(* IEC 61131-3 sources: Stat_Resistant_AI_Coding/src/plc/project/Station010, 9 files *)

(* ---- Wp100ResistanceResultStruct.st ---- *)
{attribute 'OPC.UA.DA.StructuredType':='1'}
TYPE Wp100ResistanceResultStruct :
STRUCT
  /// TRUE after SINGLE_MEAS has completed and the values below have been copied
  Valid      : BOOL;
  OutOfLimit : BOOL;
  Ok         : BOOL;
  Value      : REAL;
  Temperature : REAL;
END_STRUCT
END_TYPE

(* ---- Wp100RunResultStruct.st ---- *)
{attribute 'OPC.UA.DA.StructuredType':='1'}
TYPE Wp100RunResultStruct :
STRUCT
  /// Fixture position requested for this execution
  MeasurePos           : MeasurePsoEnum;
  /// TRUE after the requested position has passed the three-sensor one-hot check
  FixturePositionValid : BOOL;
  /// Burster resistance measurement result
  Resistance           : Wp100ResistanceResultStruct;
  /// Kistler force/stroke measurement result
  Kistler              : Wp100KistlerResultStruct;
END_STRUCT
END_TYPE

(* ---- Wp100RunSequenceResultStruct.st ---- *)
TYPE Wp100RunSequenceResultStruct :
STRUCT
  /// Result captured after the left-position atomic measurement
  Left   : Wp100RunResultStruct;
  /// Result captured after the middle-position atomic measurement
  Middle : Wp100RunResultStruct;
  /// Result captured after the right-position atomic measurement
  Right  : Wp100RunResultStruct;
END_STRUCT
END_TYPE

(* ---- AiForceTrace.gvl.st ---- *)
{attribute 'qualified_only'}
VAR_GLOBAL
  Recorder : FB_HmiForceTrace;
END_VAR

(* ---- AiWp100.gvl.st ---- *)
{attribute 'qualified_only'}
VAR_GLOBAL
  BursterProgramSelect : FB_Wp100BursterProgramSelect;
END_VAR

(* ---- FB_HmiForceTrace.st ---- *)
(* ===== OBJECT FB_HmiForceTrace ===== *)
(* ===== DECLARATION ===== *)
FUNCTION_BLOCK FB_HmiForceTrace
VAR_INPUT
  Measuring : BOOL;
  QualityGood : BOOL;
  ForceN : REAL;
END_VAR
VAR_OUTPUT
  LeftFrame : ARRAY [0..30035] OF DWORD;
  MiddleFrame : ARRAY [0..30035] OF DWORD;
  RightFrame : ARRAY [0..30035] OF DWORD;
  StatisticsFrame : ARRAY [0..209] OF DWORD;
  Published : BOOL;
  PublishedPosition : UDINT;
  Cleared : BOOL;
  Qualified : BOOL;
  DataGood : BOOL;
  SampleTime : UDINT;
END_VAR
VAR
  _stats : FB_PressForceStatistics;
  _trace : ARRAY [1..3] OF T_HmiForceBuffer;
  _stat : ARRAY [1..3,0..63] OF DWORD;
  _payloadHash : ARRAY [1..3] OF UDINT;
  _frozen : ARRAY [1..3] OF BOOL;
  _configured : BOOL;
  _guardActive : BOOL;
  _clearPending : BOOL;
  _urgent : BOOL;
  _initialized : BOOL;
  _normalEndRequested : BOOL;
  _threshold : REAL;
  _limit : REAL;
  _window : UDINT;
  _timeout : UDINT;
  _now : UDINT;
  _started : UDINT;
  _elapsed : UDINT;
  _lastSample : UDINT;
  _lastPublish : UDINT;
  _boot : UDINT;
  _cycle : UDINT;
  _acquisition : UDINT;
  _sequence : UDINT;
  _scan : UDINT;
  _sampledScan : UDINT;
  _position : UDINT;
  _state : UDINT;
  _hash : UDINT;
  _word : U_HmiForceWord;
  _p : DINT;
  _i : DINT;
  _j : DINT;
END_VAR
(* ===== IMPLEMENTATION ===== *)
// MainTask caller. HMI timing never owns acquisition or process decisions.
_now := TIME_TO_UDINT(TIME());
_scan := _scan + 1;
Published := FALSE;
Cleared := _clearPending;
_clearPending := FALSE;
IF ( NOT _initialized )
THEN
  _initialized := TRUE;
  _boot := _now;
  _urgent := TRUE;
END_IF
IF ( _state = 1 )
THEN
  IF ( NOT _guardActive )
  THEN
    Sample(ValueN := ForceN, Healthy := QualityGood, AtWork := FALSE);
  ELSIF ( ( _now - _lastSample ) > 15 )
  THEN
    // Missing cyclic guard calls must not leave a stale TRUE for the next DONE.
    DataGood := FALSE;
    Qualified := FALSE;
  END_IF
  IF ( NOT QualityGood ) OR ( NOT ( ForceN = ForceN ) ) OR
     ( ABS(ForceN) > REAL#3.402823E38 )
  THEN
    Finish(Reason := 5, LastForceN := ForceN);
  ELSIF ( NOT Measuring )
  THEN
    IF ( _normalEndRequested )
    THEN
      Finish(Reason := 2, LastForceN := ForceN);
    ELSE
      Finish(Reason := 5, LastForceN := ForceN);
    END_IF
  END_IF
END_IF
IF ( _urgent ) OR ( ( _now - _lastPublish ) >= 100 ) OR ( Cleared )
THEN
  Publish();
END_IF

(* ===== OBJECT Configure ===== *)
(* ===== DECLARATION ===== *)
METHOD PUBLIC Configure
VAR_INPUT
  ThresholdN : REAL;
  LimitN : REAL;
  WindowMs : UDINT;
  TimeoutMs : UDINT;
END_VAR
(* ===== IMPLEMENTATION ===== *)
// Once per position, before Kistler START. Changes take effect next position.
_threshold := ThresholdN;
_limit := LimitN;
_window := WindowMs;
_timeout := TimeoutMs;
_configured := TRUE;

(* ===== OBJECT BeginCycle ===== *)
(* ===== DECLARATION ===== *)
METHOD PUBLIC BeginCycle
(* ===== IMPLEMENTATION ===== *)
_cycle := _cycle + 1;
IF ( _cycle = 0 )
THEN
  _cycle := 1;
END_IF
// Only Count is authoritative. Old payload beyond Count is never displayed.
FOR _p := 1 TO 3 DO
  FOR _i := 0 TO 31 DO
    _trace[_p][_i] := 0;
  END_FOR
  FOR _i := 0 TO 63 DO
    _stat[_p,_i] := 0;
  END_FOR
  _trace[_p][1] := DWORD#2;
  _trace[_p][3] := UDINT_TO_DWORD(_cycle);
  _trace[_p][5] := DINT_TO_DWORD(_p);
  _trace[_p][16] := DWORD#6;
  _payloadHash[_p] := UDINT#2166136261;
  _frozen[_p] := FALSE;
END_FOR
_position := 0;
_state := 0;
_configured := FALSE;
_guardActive := FALSE;
Qualified := FALSE;
DataGood := FALSE;
_normalEndRequested := FALSE;
_clearPending := TRUE;
_urgent := TRUE;

(* ===== OBJECT Start ===== *)
(* ===== DECLARATION ===== *)
METHOD PUBLIC Start
VAR_INPUT
  Position : UDINT;
  InitialForceN : REAL;
END_VAR
(* ===== IMPLEMENTATION ===== *)
IF ( _state = 1 ) OR ( _cycle = 0 ) OR ( NOT _configured ) OR
   ( Position < 1 ) OR ( Position > 3 )
THEN
  RETURN;
END_IF
_acquisition := _acquisition + 1;
IF ( _acquisition = 0 )
THEN
  _acquisition := 1;
END_IF
_position := Position;
_started := TIME_TO_UDINT(TIME());
_lastSample := _started - 6;
_sampledScan := _scan - 1;
_elapsed := 0;
_state := 1;
_guardActive := FALSE;
_normalEndRequested := FALSE;
_frozen[_position] := FALSE;
_payloadHash[_position] := UDINT#2166136261;
FOR _i := 6 TO 30 DO
  _trace[_position][_i] := 0;
END_FOR
FOR _i := 0 TO 63 DO
  _stat[_position,_i] := 0;
END_FOR
_trace[_position][4] := UDINT_TO_DWORD(_acquisition);
_word.Value := _threshold;
_trace[_position][12] := _word.Bits;
_word.Value := _limit;
_trace[_position][13] := _word.Bits;
_trace[_position][14] := UDINT_TO_DWORD(_window);
_trace[_position][15] := UDINT_TO_DWORD(_timeout);
_trace[_position][16] := DWORD#6;
_stats(Enabled := FALSE);
Sample(ValueN := InitialForceN, Healthy := TRUE, AtWork := FALSE);
_urgent := TRUE;

(* ===== OBJECT Evaluate ===== *)
(* ===== DECLARATION ===== *)
METHOD PUBLIC Evaluate : BOOL
VAR_INPUT
  ValueN : REAL;
  Healthy : BOOL;
  AtWork : BOOL;
END_VAR
(* ===== IMPLEMENTATION ===== *)
// The SFC guard samples immediately before START/DONE decisions; OnCall samples
// press-down/unloading. The MainTask scan counter prevents duplicate actions;
// a 5/7 ms clock rounding pair must not skip alternate nominal 6 ms scans.
// Trace and statistics consume the SAME accepted PLC sample.
_guardActive := TRUE;
Sample(ValueN := ValueN, Healthy := Healthy, AtWork := AtWork);
Evaluate := ( _state = 1 ) AND ( DataGood ) AND ( Qualified ) AND
            ( Healthy ) AND ( AtWork ) AND ( ValueN > _threshold );

(* ===== OBJECT Sample ===== *)
(* ===== DECLARATION ===== *)
METHOD PRIVATE Sample
VAR_INPUT
  ValueN : REAL;
  Healthy : BOOL;
  AtWork : BOOL;
END_VAR
VAR
  good : BOOL;
  gap : BOOL;
  count : UDINT;
  offset : DINT;
  quality : DWORD;
END_VAR
(* ===== IMPLEMENTATION ===== *)
IF ( _state <> 1 )
THEN
  RETURN;
END_IF
_now := TIME_TO_UDINT(TIME());
good := ( Healthy ) AND ( ValueN = ValueN ) AND
        ( ABS(ValueN) <= REAL#3.402823E38 );
IF ( NOT good ) OR ( NOT AtWork ) OR ( ValueN <= _threshold )
THEN
  Qualified := FALSE;
  IF ( _guardActive ) AND ( NOT _frozen[_position] )
  THEN
    // Retain the last real window for the fault display before resetting it.
    CaptureStatistics();
    _stats(Enabled := FALSE);
  END_IF
END_IF
IF ( _sampledScan = _scan ) OR ( _now = _lastSample )
THEN
  IF ( NOT good )
  THEN
    DataGood := FALSE;
  END_IF
  RETURN;
END_IF
gap := ( ( _now - _lastSample ) > 15 );
_sampledScan := _scan;
_lastSample := _now;
SampleTime := _now;
IF ( _trace[_position][7] = 0 )
THEN
  // The actual first sampled value defines t=0 even across a millisecond tick.
  _started := _now;
END_IF
_elapsed := _now - _started;
DataGood := ( good ) AND ( NOT gap );
quality := BOOL_TO_DWORD(good);
IF ( gap )
THEN
  quality := DWORD#2;
END_IF
_trace[_position][17] := _trace[_position][17] + 1;
count := DWORD_TO_UDINT(_trace[_position][7]);
IF ( count < 10001 ) AND ( _elapsed <= 60000 )
THEN
  offset := 32 + UDINT_TO_DINT(count) * 3;
  _trace[_position][offset] := UDINT_TO_DWORD(_elapsed);
  _word.Value := ValueN;
  _trace[_position][offset+1] := _word.Bits;
  _trace[_position][offset+2] := quality;
  FOR _j := offset TO offset + 2 DO
    _payloadHash[_position] := ULINT_TO_UDINT(
      UDINT_TO_ULINT(_payloadHash[_position] XOR DWORD_TO_UDINT(_trace[_position][_j])) * ULINT#16777619);
  END_FOR
  _trace[_position][7] := UDINT_TO_DWORD(count + 1);
ELSE
  _trace[_position][8] := DWORD#1;
END_IF
IF ( _guardActive ) AND ( NOT _frozen[_position] )
THEN
  IF ( gap )
  THEN
    CaptureStatistics();
  END_IF
  _stats(Enabled := ( DataGood ) AND ( AtWork ), ForceN := ValueN,
    ThresholdN := _threshold, LimitN := _limit, WindowMs := _window, NowMs := _elapsed);
  Qualified := _stats.Qualified;
  IF ( Qualified ) AND ( _trace[_position][9] = 0 )
  THEN
    // 1-based stream number; retained capacity may already be exhausted.
    _trace[_position][9] := _trace[_position][17];
    _trace[_position][10] := UDINT_TO_DWORD(_elapsed);
    _urgent := TRUE;
  END_IF
END_IF
_word.Value := ValueN;
IF ( NOT _frozen[_position] )
THEN
  _stat[_position,5] := _word.Bits;
END_IF

(* ===== OBJECT CaptureStatistics ===== *)
(* ===== DECLARATION ===== *)
METHOD PRIVATE CaptureStatistics
VAR
  historical : BOOL;
END_VAR
(* ===== IMPLEMENTATION ===== *)
IF ( _position = 0 ) OR ( _frozen[_position] )
THEN
  RETURN;
END_IF
historical := ( _stats.Count = 0 ) AND ( _stat[_position,3] > 0 );
_stat[_position,0] := UDINT_TO_DWORD(_position);
_stat[_position,1] := UDINT_TO_DWORD(_acquisition);
_stat[_position,2] := UDINT_TO_DWORD(_state);
_stat[_position,4] := ( BOOL_TO_DWORD(DataGood) ) OR
  ( SHL(BOOL_TO_DWORD(_stats.Full),1) ) OR ( SHL(BOOL_TO_DWORD(Qualified),2) ) OR
  ( SHL(BOOL_TO_DWORD(historical),4) );
IF ( NOT historical )
THEN
_stats.SnapshotBins();
_stat[_position,3] := UDINT_TO_DWORD(_stats.Count);
_word.Value := LREAL_TO_REAL(_stats.Mean);
_stat[_position,6] := _word.Bits;
_word.Value := LREAL_TO_REAL(_stats.Sigma);
_stat[_position,7] := _word.Bits;
_word.Value := LREAL_TO_REAL(_stats.ThreeSigma);
_stat[_position,8] := _word.Bits;
_word.Value := _stats.Minimum;
_stat[_position,9] := _word.Bits;
_stat[_position,20] := _word.Bits;
_word.Value := _stats.Maximum;
_stat[_position,10] := _word.Bits;
_stat[_position,16] := UDINT_TO_DWORD(_stats.FirstMs);
_stat[_position,17] := UDINT_TO_DWORD(_stats.LastMs);
_word.Value := _stats.BinWidth;
_stat[_position,21] := _word.Bits;
_stat[_position,22] := DWORD#20;
FOR _i := 0 TO 19 DO
  _stat[_position,23 + _i] := UDINT_TO_DWORD(_stats.Bins[_i]);
END_FOR
END_IF
_stat[_position,11] := _trace[_position][12];
_stat[_position,12] := _trace[_position][13];
_stat[_position,13] := _trace[_position][14];
_stat[_position,14] := _trace[_position][15];
_stat[_position,15] := UDINT_TO_DWORD(_elapsed);
_stat[_position,18] := _trace[_position][9];
_stat[_position,19] := _trace[_position][10];
_stat[_position,43] := _trace[_position][17];
_stat[_position,44] := DWORD#6;

(* ===== OBJECT FreezeStatistics ===== *)
(* ===== DECLARATION ===== *)
METHOD PUBLIC FreezeStatistics
(* ===== IMPLEMENTATION ===== *)
IF ( _position = 0 ) OR ( _frozen[_position] )
THEN
  RETURN;
END_IF
CaptureStatistics();
_frozen[_position] := TRUE;
_stat[_position,4] := _stat[_position,4] OR DWORD#8;
_guardActive := FALSE;
_urgent := TRUE;

(* ===== OBJECT RequestEnd ===== *)
(* ===== DECLARATION ===== *)
METHOD PUBLIC RequestEnd
(* ===== IMPLEMENTATION ===== *)
IF ( _state = 1 )
THEN
  _normalEndRequested := TRUE;
END_IF

(* ===== OBJECT Finish ===== *)
(* ===== DECLARATION ===== *)
METHOD PUBLIC Finish
VAR_INPUT
  Reason : UDINT;
  LastForceN : REAL;
END_VAR
(* ===== IMPLEMENTATION ===== *)
IF ( _state <> 1 ) OR ( Reason < 2 ) OR ( Reason > 5 )
THEN
  RETURN;
END_IF
_elapsed := TIME_TO_UDINT(TIME()) - _started;
IF ( Reason <> 2 )
THEN
  Qualified := FALSE;
END_IF
IF ( Reason = 5 )
THEN
  DataGood := FALSE;
END_IF
// First terminal cause wins; cleanup cannot overwrite it.
FreezeStatistics();
_state := Reason;
_stat[_position,2] := UDINT_TO_DWORD(Reason);
IF ( Reason <> 2 )
THEN
  _stat[_position,4] := _stat[_position,4] AND NOT DWORD#4;
  _word.Value := LastForceN;
  _stat[_position,5] := _word.Bits;
END_IF
IF ( Reason = 5 )
THEN
  _stat[_position,4] := _stat[_position,4] AND NOT DWORD#1;
END_IF
_configured := FALSE;
_guardActive := FALSE;
_urgent := TRUE;

(* ===== OBJECT Publish ===== *)
(* ===== DECLARATION ===== *)
METHOD PRIVATE Publish
(* ===== IMPLEMENTATION ===== *)
_urgent := FALSE;
_lastPublish := _now;
_sequence := _sequence + 1;
IF ( _sequence = 0 )
THEN
  _sequence := 1;
END_IF
CaptureStatistics();
FOR _p := 1 TO 3 DO
  IF ( UDINT_TO_DINT(_position) = _p ) OR ( Cleared )
  THEN
    _trace[_p][0] := UDINT_TO_DWORD(_sequence);
    _trace[_p][2] := UDINT_TO_DWORD(_boot);
    IF ( UDINT_TO_DINT(_position) = _p )
    THEN
      _trace[_p][6] := UDINT_TO_DWORD(_state);
      _trace[_p][11] := UDINT_TO_DWORD(_elapsed);
    END_IF
    _hash := _payloadHash[_p];
    FOR _i := 0 TO 30 DO
      _hash := ULINT_TO_UDINT(UDINT_TO_ULINT(_hash XOR DWORD_TO_UDINT(_trace[_p][_i])) * ULINT#16777619);
    END_FOR
    _trace[_p][31] := UDINT_TO_DWORD(_hash);
    _trace[_p][30035] := _trace[_p][0];
    CASE _p OF
      1: LeftFrame := _trace[_p];
      2: MiddleFrame := _trace[_p];
      3: RightFrame := _trace[_p];
    END_CASE
  END_IF
END_FOR
StatisticsFrame[0] := UDINT_TO_DWORD(_sequence);
StatisticsFrame[1] := DWORD#2;
StatisticsFrame[2] := UDINT_TO_DWORD(_boot);
StatisticsFrame[3] := UDINT_TO_DWORD(_cycle);
StatisticsFrame[4] := UDINT_TO_DWORD(_position);
StatisticsFrame[5] := UDINT_TO_DWORD(_now);
StatisticsFrame[6] := DWORD#20;
StatisticsFrame[7] := DWORD#6;
FOR _p := 1 TO 3 DO
  FOR _i := 0 TO 63 DO
    StatisticsFrame[16 + (_p - 1) * 64 + _i] := _stat[_p,_i];
  END_FOR
END_FOR
_hash := UDINT#2166136261;
FOR _i := 0 TO 207 DO
  _hash := ULINT_TO_UDINT(UDINT_TO_ULINT(_hash XOR DWORD_TO_UDINT(StatisticsFrame[_i])) * ULINT#16777619);
END_FOR
StatisticsFrame[208] := UDINT_TO_DWORD(_hash);
StatisticsFrame[209] := StatisticsFrame[0];
PublishedPosition := _position;
Published := TRUE;

(* ---- FB_PressForceStatistics.st ---- *)
(* ===== OBJECT FB_PressForceStatistics ===== *)
(* ===== DECLARATION ===== *)
FUNCTION_BLOCK FB_PressForceStatistics
VAR_INPUT
  Enabled : BOOL;
  ForceN : REAL;
  ThresholdN : REAL;
  LimitN : REAL;
  WindowMs : UDINT;
  NowMs : UDINT;
END_VAR
VAR_OUTPUT
  Count : UDINT;
  Mean : LREAL;
  Sigma : LREAL;
  ThreeSigma : LREAL;
  Full : BOOL;
  Qualified : BOOL;
  FirstMs : UDINT;
  LastMs : UDINT;
  Minimum : REAL;
  Maximum : REAL;
  BinWidth : REAL;
  Bins : ARRAY [0..19] OF UDINT;
END_VAR
VAR
  _values : ARRAY [0..10001] OF REAL;
  _times : ARRAY [0..10001] OF UDINT;
  _head : UDINT;
  _index : UDINT;
  _next : UDINT;
  _i : UDINT;
  _bin : DINT;
  _m2 : LREAL;
  _delta : LREAL;
  _oldMean : LREAL;
  _value : LREAL;
END_VAR
(* ===== IMPLEMENTATION ===== *)
// One call per accepted PLC sample. Time-based rolling window, sample SD (n-1).
IF ( NOT Enabled ) OR ( NOT ( ForceN = ForceN ) ) OR
   ( ABS(ForceN) > REAL#3.402823E38 ) OR ( ForceN <= ThresholdN ) OR
   ( WindowMs = 0 ) OR ( WindowMs > 60000 ) OR ( LimitN <= 0 )
THEN
  Count := 0;
  _head := 0;
  Mean := 0;
  _m2 := 0;
  Sigma := 0;
  ThreeSigma := 0;
  Full := FALSE;
  Qualified := FALSE;
  FirstMs := 0;
  LastMs := 0;
  RETURN;
END_IF

// Keep one sample at/before the window start. This requires a complete time
// span, including when 1000 ms is not divisible by the 6 ms PLC task period.
WHILE ( Count > 1 ) DO
  _next := (_head + 1) MOD 10002;
  IF ( ( NowMs - _times[_next] ) < WindowMs )
  THEN
    EXIT;
  END_IF
  _value := REAL_TO_LREAL(_values[_head]);
  _oldMean := Mean;
  Mean := (UDINT_TO_LREAL(Count) * Mean - _value) / UDINT_TO_LREAL(Count - 1);
  _m2 := _m2 - (_value - _oldMean) * (_value - Mean);
  Count := Count - 1;
  _head := _next;
END_WHILE
IF ( Count >= 10002 )
THEN
  // Impossible at >=6 ms / <=60 s. Fail closed if the calling contract breaks.
  Count := 0;
  _head := 0;
  Mean := 0;
  _m2 := 0;
END_IF
_index := (_head + Count) MOD 10002;
_values[_index] := ForceN;
_times[_index] := NowMs;
Count := Count + 1;
_value := REAL_TO_LREAL(ForceN);
_delta := _value - Mean;
Mean := Mean + _delta / UDINT_TO_LREAL(Count);
_m2 := MAX(LREAL#0.0, _m2 + _delta * (_value - Mean));
FirstMs := _times[_head];
LastMs := NowMs;
Sigma := 0;
IF ( Count > 1 )
THEN
  Sigma := SQRT(_m2 / UDINT_TO_LREAL(Count - 1));
END_IF
ThreeSigma := LREAL#3.0 * Sigma;
Full := ( Count > 1 ) AND ( ( NowMs - FirstMs ) >= WindowMs );
Qualified := ( Full ) AND ( ThreeSigma < REAL_TO_LREAL(LimitN) );

(* ===== OBJECT SnapshotBins ===== *)
(* ===== DECLARATION ===== *)
METHOD PUBLIC SnapshotBins
(* ===== IMPLEMENTATION ===== *)
FOR _i := 0 TO 19 DO
  Bins[_i] := 0;
END_FOR
Minimum := 0;
Maximum := 0;
BinWidth := 0;
IF ( Count = 0 )
THEN
  RETURN;
END_IF
Minimum := _values[_head];
Maximum := Minimum;
FOR _i := 0 TO Count - 1 DO
  _index := (_head + _i) MOD 10002;
  Minimum := MIN(Minimum, _values[_index]);
  Maximum := MAX(Maximum, _values[_index]);
END_FOR
IF ( Maximum = Minimum )
THEN
  // Zero spread is displayed as a concentration marker, never a divided PDF.
  Bins[0] := Count;
  RETURN;
END_IF
BinWidth := LREAL_TO_REAL((REAL_TO_LREAL(Maximum) - REAL_TO_LREAL(Minimum)) / LREAL#20.0);
FOR _i := 0 TO Count - 1 DO
  _index := (_head + _i) MOD 10002;
  _value := (REAL_TO_LREAL(_values[_index]) - REAL_TO_LREAL(Minimum)) /
            (REAL_TO_LREAL(Maximum) - REAL_TO_LREAL(Minimum)) * LREAL#20.0;
  _bin := LIMIT(0, LREAL_TO_DINT(TRUNC(_value)), 19);
  Bins[_bin] := Bins[_bin] + 1;
END_FOR

(* ---- FB_Wp100BursterProgramSelect.st ---- *)
(*
  Canonical AI-owned POU. Same-owner adapter for the existing SFC API.
  No socket here: all protocol operations belong to Peripherals._Burster2316.
*)
(* ===== DECLARATION ===== *)
FUNCTION_BLOCK FB_Wp100BursterProgramSelect
VAR_INPUT
  Execute : BOOL;
  ProgramNo : INT;
END_VAR
VAR_OUTPUT
  Busy : BOOL;
  Done : BOOL;
  Error : BOOL;
  ErrorCode : DINT;
  LastSocketError : OpconDeviceError;
END_VAR
VAR
  _state : USINT; // 0=idle, 10=Open, 20=select, 90=cancel, 100=done, 200=error
  _requestedProgramNo : INT;
  _ret : DINT;
END_VAR

(* ===== IMPLEMENTATION ===== *)
// Only N045 (with the standard Unit READY/Execute=FALSE) starts selection.
// Resetting the adapter AFTER Done must not close a later Unit measurement.
IF ( NOT Execute )
THEN
  Done := FALSE;
  IF ( _state = 0 ) OR ( _state = 100 ) OR ( _state = 200 )
  THEN
    _state := 0;
    Busy := FALSE;
    Error := FALSE;
    RETURN;
  END_IF
  _state := 90;
END_IF

IF ( Execute ) AND
   ( ( _state = 10 ) OR ( _state = 20 ) ) AND
   ( ProgramNo <> _requestedProgramNo )
THEN
  IF ( ErrorCode = 0 ) THEN ErrorCode := 1503; END_IF
  Error := TRUE;
  _state := 90;
END_IF

CASE _state OF
  0:
    Busy := TRUE;
    Done := FALSE;
    Error := FALSE;
    ErrorCode := 0;
    _ret := RUNNING;
    OpconMemSet(ADR(LastSocketError), 0, SIZEOF(LastSocketError));
    IF ( ProgramNo < 0 ) OR ( ProgramNo > 15 )
    THEN
      ErrorCode := 1501;
      Error := TRUE;
      Busy := FALSE;
      _state := 200;
    ELSE
      _requestedProgramNo := ProgramNo;
      _state := 10;
    END_IF
  10:
    _ret := Peripherals._Burster2316.Open();
    IF ( _ret = OK ) THEN _state := 20; END_IF
  20:
    _ret := Peripherals._Burster2316.SelectProgram(ProgramNo := _requestedProgramNo);
    IF ( _ret = OK )
    THEN
      Busy := FALSE;
      Done := TRUE;
      _state := 100;
    END_IF
  90:
    // Continue only cancellation of our Open/Select call. If the Unit already
    // owns a measurement/error-clear, never replace it with a second Reset.
    IF ( Peripherals._Burster2316.Operation = 0 ) OR
       ( Peripherals._Burster2316.Operation = 1 ) OR
       ( Peripherals._Burster2316.Operation = 2 ) OR
       ( Peripherals._Burster2316.Operation = 9 )
    THEN
      _ret := Peripherals._Burster2316.Reset();
      IF ( _ret <> RUNNING )
      THEN
        IF ( _ret < OK )
        THEN
          IF ( ErrorCode = 0 )
          THEN
            ErrorCode := Peripherals._Burster2316.ErrorCode;
            IF ( ErrorCode = 0 ) THEN ErrorCode := 1502; END_IF
            LastSocketError := Peripherals._Burster2316.LastError;
          END_IF
          Error := TRUE;
        END_IF
        Busy := FALSE;
        IF ( Error ) THEN _state := 200; ELSE _state := 0; END_IF
      END_IF
    ELSE
      IF ( ErrorCode = 0 ) THEN ErrorCode := 1502; END_IF
      Error := TRUE;
      Busy := FALSE;
      _state := 200;
    END_IF
  100:
    ; // Hold Done until Execute falls; never recall the program here.
  200:
    ; // Preserve first fault until Execute falls; no automatic reconnect.
END_CASE

IF ( ( _state = 10 ) OR ( _state = 20 ) ) AND
   ( _ret < OK )
THEN
  IF ( ErrorCode = 0 )
  THEN
    ErrorCode := Peripherals._Burster2316.ErrorCode;
    IF ( ErrorCode = 0 ) THEN ErrorCode := 1502; END_IF
    LastSocketError := Peripherals._Burster2316.LastError;
  END_IF
  Error := TRUE;
  Done := FALSE;
  Busy := TRUE;
  _state := 90; // Continue the pending owner's cleanup even after SFC stops.
END_IF

(* ---- Wp100KistlerResultStruct.st ---- *)
{attribute 'OPC.UA.DA.StructuredType':='1'}
TYPE Wp100KistlerResultStruct :
STRUCT
  /// TRUE after the MEASURE command has completed and the values below have been copied
  Valid     : BOOL;
  Ok        : BOOL;
  Nok       : BOOL;
  NoPass    : BOOL;
  ProgramNo : BYTE;
  Force     : REAL;
  Stroke    : REAL;
END_STRUCT
END_TYPE
